// Implicitly generated code : DO NOT EDIT
FUNCTION CheckDivReal : REAL
VAR_INPUT
    divisor:REAL;
END_VAR


// Implicitly generated code : Only an Implementation suggestion
{noflow}
IF divisor = 0 THEN
    CheckDivReal:=1;
ELSE
    CheckDivReal:=divisor;
END_IF;
{flow}

END_FUNCTION

(* stored: Version 1.1.0.1
   POU CheckDivReal: Id {642e0c23-2413-4ca5-8e92-8ce69fff3a96}, SpecialFunc CheckDivReal32 *)
